{attribute 'qualified_only'}
{attribute 'strict'}
TYPE ERetCode_t :
(
	eRetFailed := 0,
	eRetBusy,
	eRetDone
);
END_TYPE

(* stored: Version 1.1.0.1, ProductVersion 3.1.4024.9
   DUT ERetCode_t: Id {f174652a-7676-462f-840c-197fcbddb504} *)
